// TIA Portal V17 export
// export: Created 2023-04-07T09:30:33.3999419Z, ExportSetting WithDefaults, DisplayName Totally Integrated Automation Portal, DisplayVersion V17 Update 4, DisplayName TIA Portal Openness, DisplayVersion V17 Update 4, DisplayName TIA Portal Version Control Interface, DisplayVersion V17, DisplayName STEP 7 Professional, DisplayVersion V17 Update 4, DisplayName STEP 7 Safety, DisplayVersion V17, DisplayName WinCC Professional, DisplayVersion V17 Update 4
FUNCTION "PCS Faults_1" : Void   // FC43, LAD
{ S7_Optimized_Access := 'TRUE' }
VERSION : 0.1
// stored: AutoNumber false, IsIECCheckEnabled false, SetENOAutomatically false, UDAEnableTagReadback false
   VAR_TEMP
      wMF1 : Word;
      wMF2 : Word;
      wMF3 : Word;
      wMF4 : Word;
      wMW1 : Word;
      wMW2 : Word;
      wMW3 : Word;
      wMW4 : Word;
   END_VAR
   VAR_TEMP   // added for the SCL form of the ladder/FBD networks
      _w1 : Bool;
      _w2 : Bool;
      _w3 : Bool;
      _w4 : Bool;
   END_VAR
BEGIN

REGION Network 1: Inverter Faults
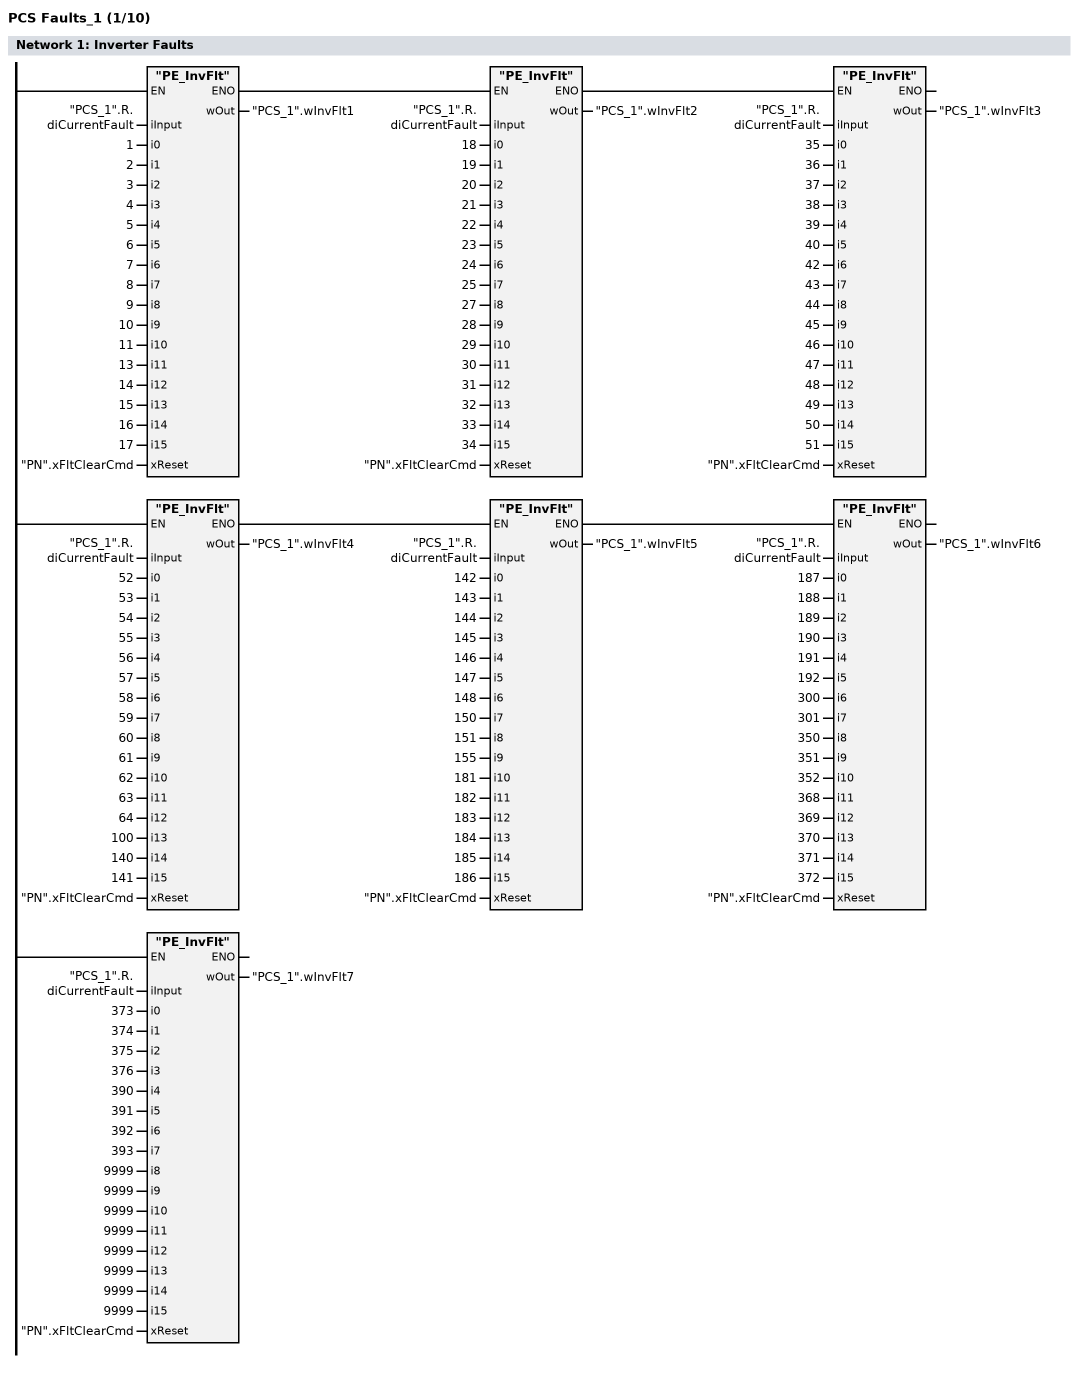
   RUNG wire#powerrail
      "PE_InvFlt"(iInput := "PCS_1".R.diCurrentFault, i0 := 1, i1 := 2, i2 := 3, i3 := 4, i4 := 5, i5 := 6, i6 := 7, i7 := 8, i8 := 9, i9 := 10, i10 := 11, i11 := 13, i12 := 14, i13 := 15, i14 := 16, i15 := 17, xReset := "PN".xFltClearCmd, wOut => "PCS_1".wInvFlt1)
      "PE_InvFlt"(iInput := "PCS_1".R.diCurrentFault, i0 := 18, i1 := 19, i2 := 20, i3 := 21, i4 := 22, i5 := 23, i6 := 24, i7 := 25, i8 := 27, i9 := 28, i10 := 29, i11 := 30, i12 := 31, i13 := 32, i14 := 33, i15 := 34, xReset := "PN".xFltClearCmd, wOut => "PCS_1".wInvFlt2)
      "PE_InvFlt"(iInput := "PCS_1".R.diCurrentFault, i0 := 35, i1 := 36, i2 := 37, i3 := 38, i4 := 39, i5 := 40, i6 := 42, i7 := 43, i8 := 44, i9 := 45, i10 := 46, i11 := 47, i12 := 48, i13 := 49, i14 := 50, i15 := 51, xReset := "PN".xFltClearCmd, wOut => "PCS_1".wInvFlt3)
   END_RUNG
   RUNG wire#powerrail
      "PE_InvFlt"(iInput := "PCS_1".R.diCurrentFault, i0 := 52, i1 := 53, i2 := 54, i3 := 55, i4 := 56, i5 := 57, i6 := 58, i7 := 59, i8 := 60, i9 := 61, i10 := 62, i11 := 63, i12 := 64, i13 := 100, i14 := 140, i15 := 141, xReset := "PN".xFltClearCmd, wOut => "PCS_1".wInvFlt4)
      "PE_InvFlt"(iInput := "PCS_1".R.diCurrentFault, i0 := 142, i1 := 143, i2 := 144, i3 := 145, i4 := 146, i5 := 147, i6 := 148, i7 := 150, i8 := 151, i9 := 155, i10 := 181, i11 := 182, i12 := 183, i13 := 184, i14 := 185, i15 := 186, xReset := "PN".xFltClearCmd, wOut => "PCS_1".wInvFlt5)
      "PE_InvFlt"(iInput := "PCS_1".R.diCurrentFault, i0 := 187, i1 := 188, i2 := 189, i3 := 190, i4 := 191, i5 := 192, i6 := 300, i7 := 301, i8 := 350, i9 := 351, i10 := 352, i11 := 368, i12 := 369, i13 := 370, i14 := 371, i15 := 372, xReset := "PN".xFltClearCmd, wOut => "PCS_1".wInvFlt6)
   END_RUNG
   RUNG wire#powerrail
      "PE_InvFlt"(iInput := "PCS_1".R.diCurrentFault, i0 := 373, i1 := 374, i2 := 375, i3 := 376, i4 := 390, i5 := 391, i6 := 392, i7 := 393, i8 := 9999, i9 := 9999, i10 := 9999, i11 := 9999, i12 := 9999, i13 := 9999, i14 := 9999, i15 := 9999, xReset := "PN".xFltClearCmd, wOut => "PCS_1".wInvFlt7)
   END_RUNG
   // the same network as SCL:
   "PE_InvFlt"(iInput := "PCS_1".R.diCurrentFault,
               i0 := 1,
               i1 := 2,
               i2 := 3,
               i3 := 4,
               i4 := 5,
               i5 := 6,
               i6 := 7,
               i7 := 8,
               i8 := 9,
               i9 := 10,
               i10 := 11,
               i11 := 13,
               i12 := 14,
               i13 := 15,
               i14 := 16,
               i15 := 17,
               xReset := "PN".xFltClearCmd,
               wOut => "PCS_1".wInvFlt1,
               ENO => #_w1);
   "PE_InvFlt"(EN := #_w1,
               iInput := "PCS_1".R.diCurrentFault,
               i0 := 18,
               i1 := 19,
               i2 := 20,
               i3 := 21,
               i4 := 22,
               i5 := 23,
               i6 := 24,
               i7 := 25,
               i8 := 27,
               i9 := 28,
               i10 := 29,
               i11 := 30,
               i12 := 31,
               i13 := 32,
               i14 := 33,
               i15 := 34,
               xReset := "PN".xFltClearCmd,
               wOut => "PCS_1".wInvFlt2,
               ENO => #_w2);
   IF #_w2 THEN
       "PE_InvFlt"(iInput := "PCS_1".R.diCurrentFault,
                   i0 := 35,
                   i1 := 36,
                   i2 := 37,
                   i3 := 38,
                   i4 := 39,
                   i5 := 40,
                   i6 := 42,
                   i7 := 43,
                   i8 := 44,
                   i9 := 45,
                   i10 := 46,
                   i11 := 47,
                   i12 := 48,
                   i13 := 49,
                   i14 := 50,
                   i15 := 51,
                   xReset := "PN".xFltClearCmd,
                   wOut => "PCS_1".wInvFlt3);
   END_IF;
   "PE_InvFlt"(iInput := "PCS_1".R.diCurrentFault,
               i0 := 52,
               i1 := 53,
               i2 := 54,
               i3 := 55,
               i4 := 56,
               i5 := 57,
               i6 := 58,
               i7 := 59,
               i8 := 60,
               i9 := 61,
               i10 := 62,
               i11 := 63,
               i12 := 64,
               i13 := 100,
               i14 := 140,
               i15 := 141,
               xReset := "PN".xFltClearCmd,
               wOut => "PCS_1".wInvFlt4,
               ENO => #_w3);
   "PE_InvFlt"(EN := #_w3,
               iInput := "PCS_1".R.diCurrentFault,
               i0 := 142,
               i1 := 143,
               i2 := 144,
               i3 := 145,
               i4 := 146,
               i5 := 147,
               i6 := 148,
               i7 := 150,
               i8 := 151,
               i9 := 155,
               i10 := 181,
               i11 := 182,
               i12 := 183,
               i13 := 184,
               i14 := 185,
               i15 := 186,
               xReset := "PN".xFltClearCmd,
               wOut => "PCS_1".wInvFlt5,
               ENO => #_w4);
   IF #_w4 THEN
       "PE_InvFlt"(iInput := "PCS_1".R.diCurrentFault,
                   i0 := 187,
                   i1 := 188,
                   i2 := 189,
                   i3 := 190,
                   i4 := 191,
                   i5 := 192,
                   i6 := 300,
                   i7 := 301,
                   i8 := 350,
                   i9 := 351,
                   i10 := 352,
                   i11 := 368,
                   i12 := 369,
                   i13 := 370,
                   i14 := 371,
                   i15 := 372,
                   xReset := "PN".xFltClearCmd,
                   wOut => "PCS_1".wInvFlt6);
   END_IF;
   "PE_InvFlt"(iInput := "PCS_1".R.diCurrentFault,
               i0 := 373,
               i1 := 374,
               i2 := 375,
               i3 := 376,
               i4 := 390,
               i5 := 391,
               i6 := 392,
               i7 := 393,
               i8 := 9999,
               i9 := 9999,
               i10 := 9999,
               i11 := 9999,
               i12 := 9999,
               i13 := 9999,
               i14 := 9999,
               i15 := 9999,
               xReset := "PN".xFltClearCmd,
               wOut => "PCS_1".wInvFlt7);
END_REGION

REGION Network 2: Inverter Warning
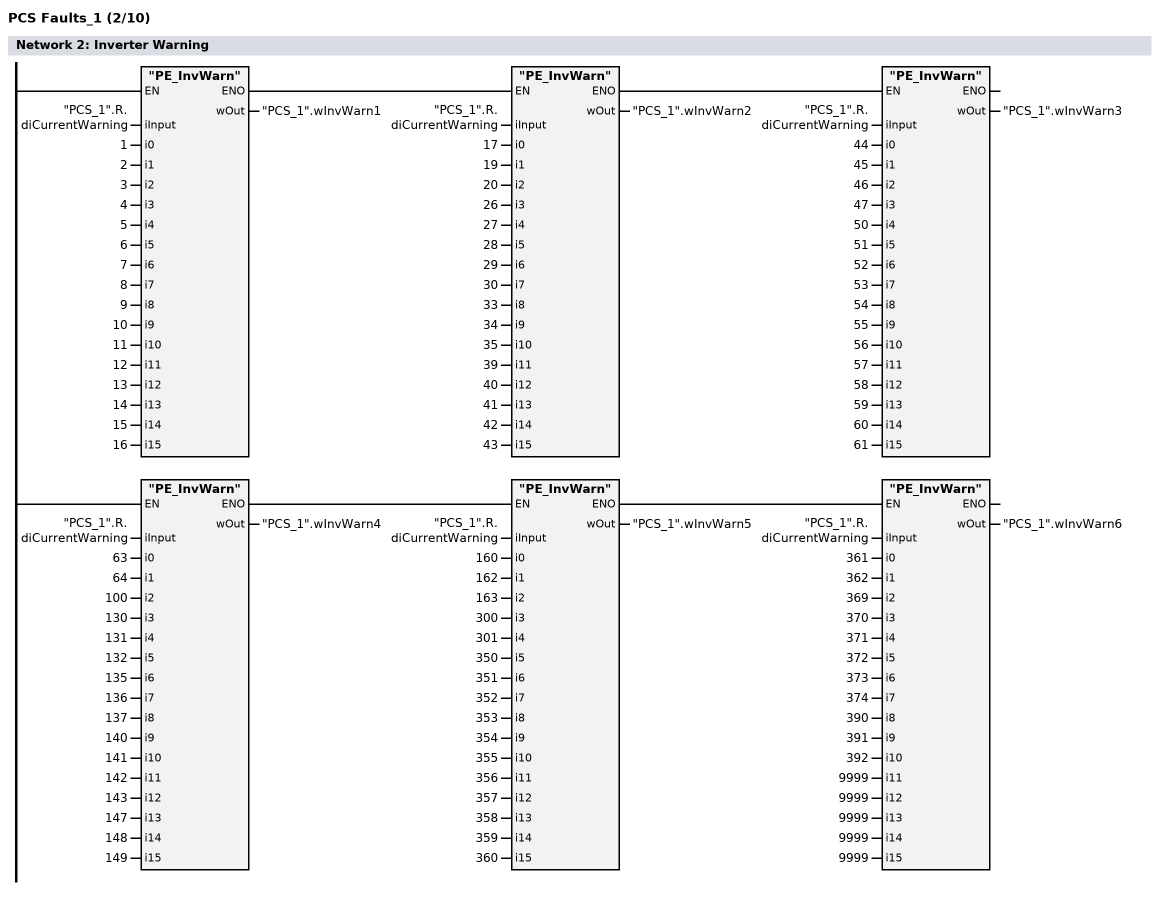
   RUNG wire#powerrail
      "PE_InvWarn"(iInput := "PCS_1".R.diCurrentWarning, i0 := 1, i1 := 2, i2 := 3, i3 := 4, i4 := 5, i5 := 6, i6 := 7, i7 := 8, i8 := 9, i9 := 10, i10 := 11, i11 := 12, i12 := 13, i13 := 14, i14 := 15, i15 := 16, wOut => "PCS_1".wInvWarn1)
      "PE_InvWarn"(iInput := "PCS_1".R.diCurrentWarning, i0 := 17, i1 := 19, i2 := 20, i3 := 26, i4 := 27, i5 := 28, i6 := 29, i7 := 30, i8 := 33, i9 := 34, i10 := 35, i11 := 39, i12 := 40, i13 := 41, i14 := 42, i15 := 43, wOut => "PCS_1".wInvWarn2)
      "PE_InvWarn"(iInput := "PCS_1".R.diCurrentWarning, i0 := 44, i1 := 45, i2 := 46, i3 := 47, i4 := 50, i5 := 51, i6 := 52, i7 := 53, i8 := 54, i9 := 55, i10 := 56, i11 := 57, i12 := 58, i13 := 59, i14 := 60, i15 := 61, wOut => "PCS_1".wInvWarn3)
   END_RUNG
   RUNG wire#powerrail
      "PE_InvWarn"(iInput := "PCS_1".R.diCurrentWarning, i0 := 63, i1 := 64, i2 := 100, i3 := 130, i4 := 131, i5 := 132, i6 := 135, i7 := 136, i8 := 137, i9 := 140, i10 := 141, i11 := 142, i12 := 143, i13 := 147, i14 := 148, i15 := 149, wOut => "PCS_1".wInvWarn4)
      "PE_InvWarn"(iInput := "PCS_1".R.diCurrentWarning, i0 := 160, i1 := 162, i2 := 163, i3 := 300, i4 := 301, i5 := 350, i6 := 351, i7 := 352, i8 := 353, i9 := 354, i10 := 355, i11 := 356, i12 := 357, i13 := 358, i14 := 359, i15 := 360, wOut => "PCS_1".wInvWarn5)
      "PE_InvWarn"(iInput := "PCS_1".R.diCurrentWarning, i0 := 361, i1 := 362, i2 := 369, i3 := 370, i4 := 371, i5 := 372, i6 := 373, i7 := 374, i8 := 390, i9 := 391, i10 := 392, i11 := 9999, i12 := 9999, i13 := 9999, i14 := 9999, i15 := 9999, wOut => "PCS_1".wInvWarn6)
   END_RUNG
   // the same network as SCL:
   "PE_InvWarn"(iInput := "PCS_1".R.diCurrentWarning,
                i0 := 1,
                i1 := 2,
                i2 := 3,
                i3 := 4,
                i4 := 5,
                i5 := 6,
                i6 := 7,
                i7 := 8,
                i8 := 9,
                i9 := 10,
                i10 := 11,
                i11 := 12,
                i12 := 13,
                i13 := 14,
                i14 := 15,
                i15 := 16,
                wOut => "PCS_1".wInvWarn1,
                ENO => #_w1);
   "PE_InvWarn"(EN := #_w1,
                iInput := "PCS_1".R.diCurrentWarning,
                i0 := 17,
                i1 := 19,
                i2 := 20,
                i3 := 26,
                i4 := 27,
                i5 := 28,
                i6 := 29,
                i7 := 30,
                i8 := 33,
                i9 := 34,
                i10 := 35,
                i11 := 39,
                i12 := 40,
                i13 := 41,
                i14 := 42,
                i15 := 43,
                wOut => "PCS_1".wInvWarn2,
                ENO => #_w2);
   IF #_w2 THEN
       "PE_InvWarn"(iInput := "PCS_1".R.diCurrentWarning,
                    i0 := 44,
                    i1 := 45,
                    i2 := 46,
                    i3 := 47,
                    i4 := 50,
                    i5 := 51,
                    i6 := 52,
                    i7 := 53,
                    i8 := 54,
                    i9 := 55,
                    i10 := 56,
                    i11 := 57,
                    i12 := 58,
                    i13 := 59,
                    i14 := 60,
                    i15 := 61,
                    wOut => "PCS_1".wInvWarn3);
   END_IF;
   "PE_InvWarn"(iInput := "PCS_1".R.diCurrentWarning,
                i0 := 63,
                i1 := 64,
                i2 := 100,
                i3 := 130,
                i4 := 131,
                i5 := 132,
                i6 := 135,
                i7 := 136,
                i8 := 137,
                i9 := 140,
                i10 := 141,
                i11 := 142,
                i12 := 143,
                i13 := 147,
                i14 := 148,
                i15 := 149,
                wOut => "PCS_1".wInvWarn4,
                ENO => #_w3);
   "PE_InvWarn"(EN := #_w3,
                iInput := "PCS_1".R.diCurrentWarning,
                i0 := 160,
                i1 := 162,
                i2 := 163,
                i3 := 300,
                i4 := 301,
                i5 := 350,
                i6 := 351,
                i7 := 352,
                i8 := 353,
                i9 := 354,
                i10 := 355,
                i11 := 356,
                i12 := 357,
                i13 := 358,
                i14 := 359,
                i15 := 360,
                wOut => "PCS_1".wInvWarn5,
                ENO => #_w4);
   IF #_w4 THEN
       "PE_InvWarn"(iInput := "PCS_1".R.diCurrentWarning,
                    i0 := 361,
                    i1 := 362,
                    i2 := 369,
                    i3 := 370,
                    i4 := 371,
                    i5 := 372,
                    i6 := 373,
                    i7 := 374,
                    i8 := 390,
                    i9 := 391,
                    i10 := 392,
                    i11 := 9999,
                    i12 := 9999,
                    i13 := 9999,
                    i14 := 9999,
                    i15 := 9999,
                    wOut => "PCS_1".wInvWarn6);
   END_IF;
END_REGION

REGION Network 3: Module Faults
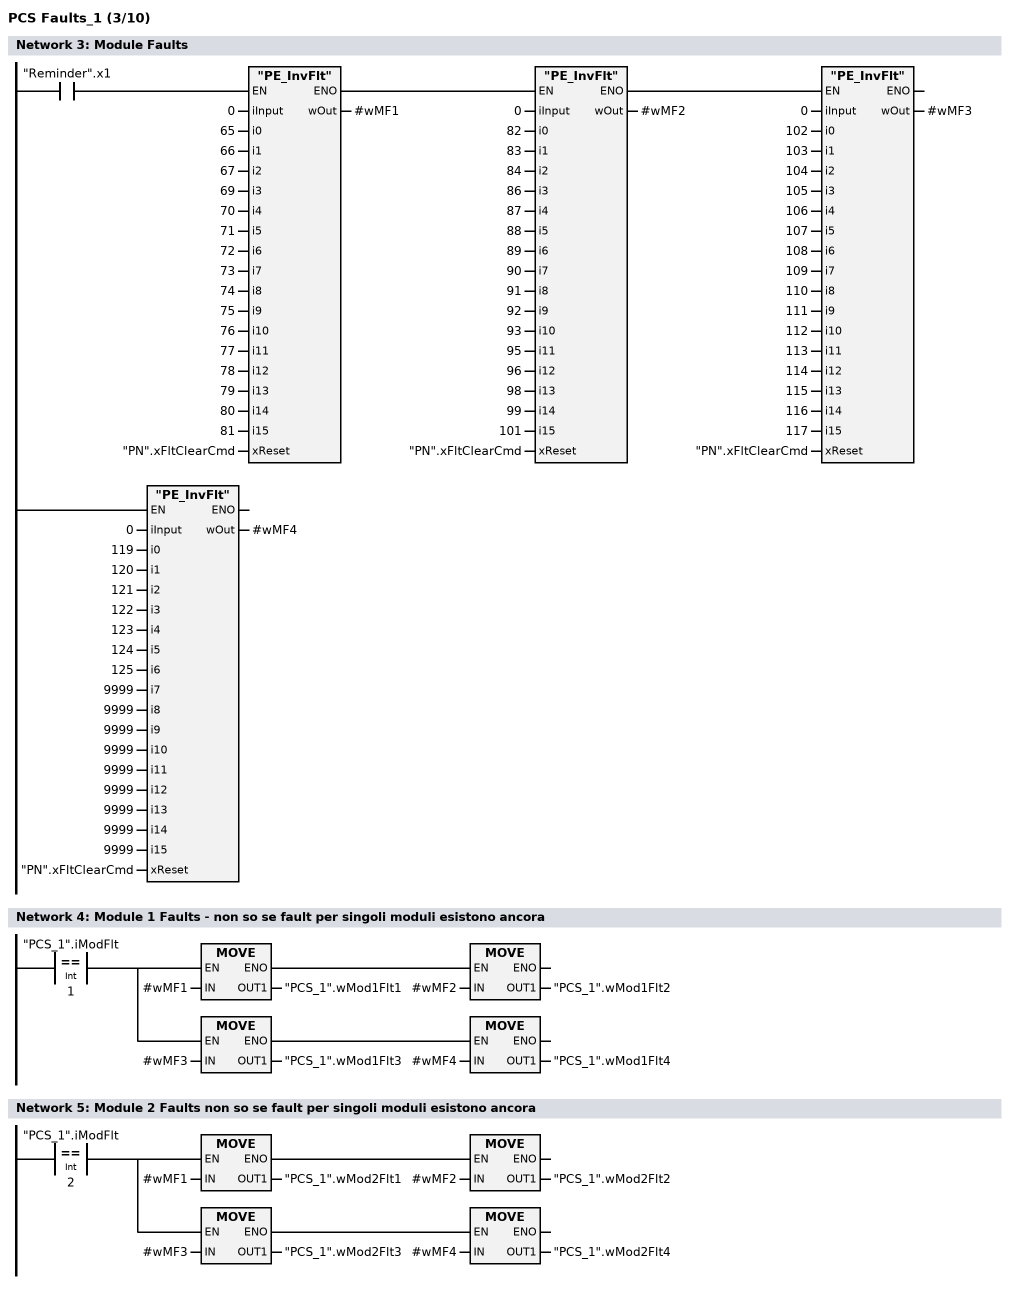
   RUNG wire#powerrail
      Contact( "Reminder".x1 )
      "PE_InvFlt"(iInput := 0, i0 := 65, i1 := 66, i2 := 67, i3 := 69, i4 := 70, i5 := 71, i6 := 72, i7 := 73, i8 := 74, i9 := 75, i10 := 76, i11 := 77, i12 := 78, i13 := 79, i14 := 80, i15 := 81, xReset := "PN".xFltClearCmd, wOut => #wMF1)
      "PE_InvFlt"(iInput := 0, i0 := 82, i1 := 83, i2 := 84, i3 := 86, i4 := 87, i5 := 88, i6 := 89, i7 := 90, i8 := 91, i9 := 92, i10 := 93, i11 := 95, i12 := 96, i13 := 98, i14 := 99, i15 := 101, xReset := "PN".xFltClearCmd, wOut => #wMF2)
      "PE_InvFlt"(iInput := 0, i0 := 102, i1 := 103, i2 := 104, i3 := 105, i4 := 106, i5 := 107, i6 := 108, i7 := 109, i8 := 110, i9 := 111, i10 := 112, i11 := 113, i12 := 114, i13 := 115, i14 := 116, i15 := 117, xReset := "PN".xFltClearCmd, wOut => #wMF3)
   END_RUNG
   RUNG wire#powerrail
      "PE_InvFlt"(iInput := 0, i0 := 119, i1 := 120, i2 := 121, i3 := 122, i4 := 123, i5 := 124, i6 := 125, i7 := 9999, i8 := 9999, i9 := 9999, i10 := 9999, i11 := 9999, i12 := 9999, i13 := 9999, i14 := 9999, i15 := 9999, xReset := "PN".xFltClearCmd, wOut => #wMF4)
   END_RUNG
   // the same network as SCL:
   "PE_InvFlt"(EN := "Reminder".x1,
               iInput := 0,
               i0 := 65,
               i1 := 66,
               i2 := 67,
               i3 := 69,
               i4 := 70,
               i5 := 71,
               i6 := 72,
               i7 := 73,
               i8 := 74,
               i9 := 75,
               i10 := 76,
               i11 := 77,
               i12 := 78,
               i13 := 79,
               i14 := 80,
               i15 := 81,
               xReset := "PN".xFltClearCmd,
               wOut => #wMF1,
               ENO => #_w1);
   "PE_InvFlt"(EN := #_w1,
               iInput := 0,
               i0 := 82,
               i1 := 83,
               i2 := 84,
               i3 := 86,
               i4 := 87,
               i5 := 88,
               i6 := 89,
               i7 := 90,
               i8 := 91,
               i9 := 92,
               i10 := 93,
               i11 := 95,
               i12 := 96,
               i13 := 98,
               i14 := 99,
               i15 := 101,
               xReset := "PN".xFltClearCmd,
               wOut => #wMF2,
               ENO => #_w2);
   IF #_w2 THEN
       "PE_InvFlt"(iInput := 0,
                   i0 := 102,
                   i1 := 103,
                   i2 := 104,
                   i3 := 105,
                   i4 := 106,
                   i5 := 107,
                   i6 := 108,
                   i7 := 109,
                   i8 := 110,
                   i9 := 111,
                   i10 := 112,
                   i11 := 113,
                   i12 := 114,
                   i13 := 115,
                   i14 := 116,
                   i15 := 117,
                   xReset := "PN".xFltClearCmd,
                   wOut => #wMF3);
   END_IF;
   "PE_InvFlt"(iInput := 0,
               i0 := 119,
               i1 := 120,
               i2 := 121,
               i3 := 122,
               i4 := 123,
               i5 := 124,
               i6 := 125,
               i7 := 9999,
               i8 := 9999,
               i9 := 9999,
               i10 := 9999,
               i11 := 9999,
               i12 := 9999,
               i13 := 9999,
               i14 := 9999,
               i15 := 9999,
               xReset := "PN".xFltClearCmd,
               wOut => #wMF4);
END_REGION

REGION Network 4: Module 1 Faults - non so se fault per singoli moduli esistono ancora
   RUNG wire#powerrail
      { S7_Templates := "SrcType := Int" } EQ_Contact(in1 := "PCS_1".iModFlt, in2 := 1)
      wire#w1
      Move(in := #wMF1, out1 => "PCS_1".wMod1Flt1)
      Move(in := #wMF2, out1 => "PCS_1".wMod1Flt2)
   END_RUNG
   RUNG wire#w1
      Move(in := #wMF3, out1 => "PCS_1".wMod1Flt3)
      Move(in := #wMF4, out1 => "PCS_1".wMod1Flt4)
   END_RUNG
   // the same network as SCL:
   IF "PCS_1".iModFlt = 1 THEN
       "PCS_1".wMod1Flt1 := #wMF1;
       "PCS_1".wMod1Flt2 := #wMF2;
       "PCS_1".wMod1Flt3 := #wMF3;
       "PCS_1".wMod1Flt4 := #wMF4;
   END_IF;
END_REGION

REGION Network 5: Module 2 Faults non so se fault per singoli moduli esistono ancora
   RUNG wire#powerrail
      { S7_Templates := "SrcType := Int" } EQ_Contact(in1 := "PCS_1".iModFlt, in2 := 2)
      wire#w1
      Move(in := #wMF1, out1 => "PCS_1".wMod2Flt1)
      Move(in := #wMF2, out1 => "PCS_1".wMod2Flt2)
   END_RUNG
   RUNG wire#w1
      Move(in := #wMF3, out1 => "PCS_1".wMod2Flt3)
      Move(in := #wMF4, out1 => "PCS_1".wMod2Flt4)
   END_RUNG
   // the same network as SCL:
   IF "PCS_1".iModFlt = 2 THEN
       "PCS_1".wMod2Flt1 := #wMF1;
       "PCS_1".wMod2Flt2 := #wMF2;
       "PCS_1".wMod2Flt3 := #wMF3;
       "PCS_1".wMod2Flt4 := #wMF4;
   END_IF;
END_REGION

REGION Network 6: Module 3 Faults
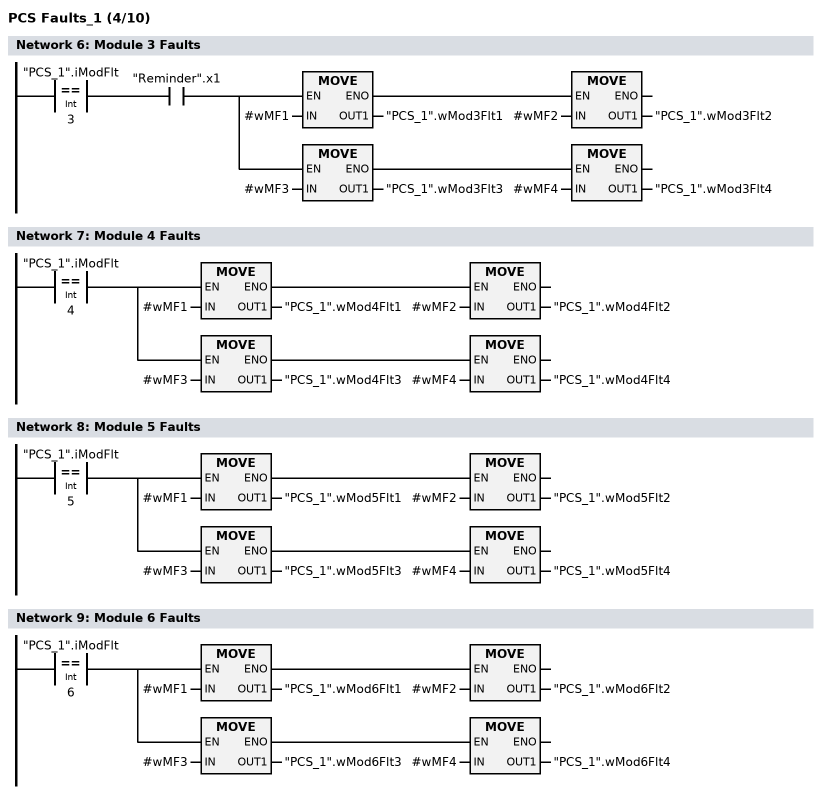
   RUNG wire#powerrail
      { S7_Templates := "SrcType := Int" } EQ_Contact(in1 := "PCS_1".iModFlt, in2 := 3)
      Contact( "Reminder".x1 )
      wire#w1
      Move(in := #wMF1, out1 => "PCS_1".wMod3Flt1)
      Move(in := #wMF2, out1 => "PCS_1".wMod3Flt2)
   END_RUNG
   RUNG wire#w1
      Move(in := #wMF3, out1 => "PCS_1".wMod3Flt3)
      Move(in := #wMF4, out1 => "PCS_1".wMod3Flt4)
   END_RUNG
   // the same network as SCL:
   IF ("PCS_1".iModFlt = 3) AND "Reminder".x1 THEN
       "PCS_1".wMod3Flt1 := #wMF1;
       "PCS_1".wMod3Flt2 := #wMF2;
       "PCS_1".wMod3Flt3 := #wMF3;
       "PCS_1".wMod3Flt4 := #wMF4;
   END_IF;
END_REGION

REGION Network 7: Module 4 Faults
   RUNG wire#powerrail
      { S7_Templates := "SrcType := Int" } EQ_Contact(in1 := "PCS_1".iModFlt, in2 := 4)
      wire#w1
      Move(in := #wMF1, out1 => "PCS_1".wMod4Flt1)
      Move(in := #wMF2, out1 => "PCS_1".wMod4Flt2)
   END_RUNG
   RUNG wire#w1
      Move(in := #wMF3, out1 => "PCS_1".wMod4Flt3)
      Move(in := #wMF4, out1 => "PCS_1".wMod4Flt4)
   END_RUNG
   // the same network as SCL:
   IF "PCS_1".iModFlt = 4 THEN
       "PCS_1".wMod4Flt1 := #wMF1;
       "PCS_1".wMod4Flt2 := #wMF2;
       "PCS_1".wMod4Flt3 := #wMF3;
       "PCS_1".wMod4Flt4 := #wMF4;
   END_IF;
END_REGION

REGION Network 8: Module 5 Faults
   RUNG wire#powerrail
      { S7_Templates := "SrcType := Int" } EQ_Contact(in1 := "PCS_1".iModFlt, in2 := 5)
      wire#w1
      Move(in := #wMF1, out1 => "PCS_1".wMod5Flt1)
      Move(in := #wMF2, out1 => "PCS_1".wMod5Flt2)
   END_RUNG
   RUNG wire#w1
      Move(in := #wMF3, out1 => "PCS_1".wMod5Flt3)
      Move(in := #wMF4, out1 => "PCS_1".wMod5Flt4)
   END_RUNG
   // the same network as SCL:
   IF "PCS_1".iModFlt = 5 THEN
       "PCS_1".wMod5Flt1 := #wMF1;
       "PCS_1".wMod5Flt2 := #wMF2;
       "PCS_1".wMod5Flt3 := #wMF3;
       "PCS_1".wMod5Flt4 := #wMF4;
   END_IF;
END_REGION

REGION Network 9: Module 6 Faults
   RUNG wire#powerrail
      { S7_Templates := "SrcType := Int" } EQ_Contact(in1 := "PCS_1".iModFlt, in2 := 6)
      wire#w1
      Move(in := #wMF1, out1 => "PCS_1".wMod6Flt1)
      Move(in := #wMF2, out1 => "PCS_1".wMod6Flt2)
   END_RUNG
   RUNG wire#w1
      Move(in := #wMF3, out1 => "PCS_1".wMod6Flt3)
      Move(in := #wMF4, out1 => "PCS_1".wMod6Flt4)
   END_RUNG
   // the same network as SCL:
   IF "PCS_1".iModFlt = 6 THEN
       "PCS_1".wMod6Flt1 := #wMF1;
       "PCS_1".wMod6Flt2 := #wMF2;
       "PCS_1".wMod6Flt3 := #wMF3;
       "PCS_1".wMod6Flt4 := #wMF4;
   END_IF;
END_REGION

REGION Network 10: Module Warnings
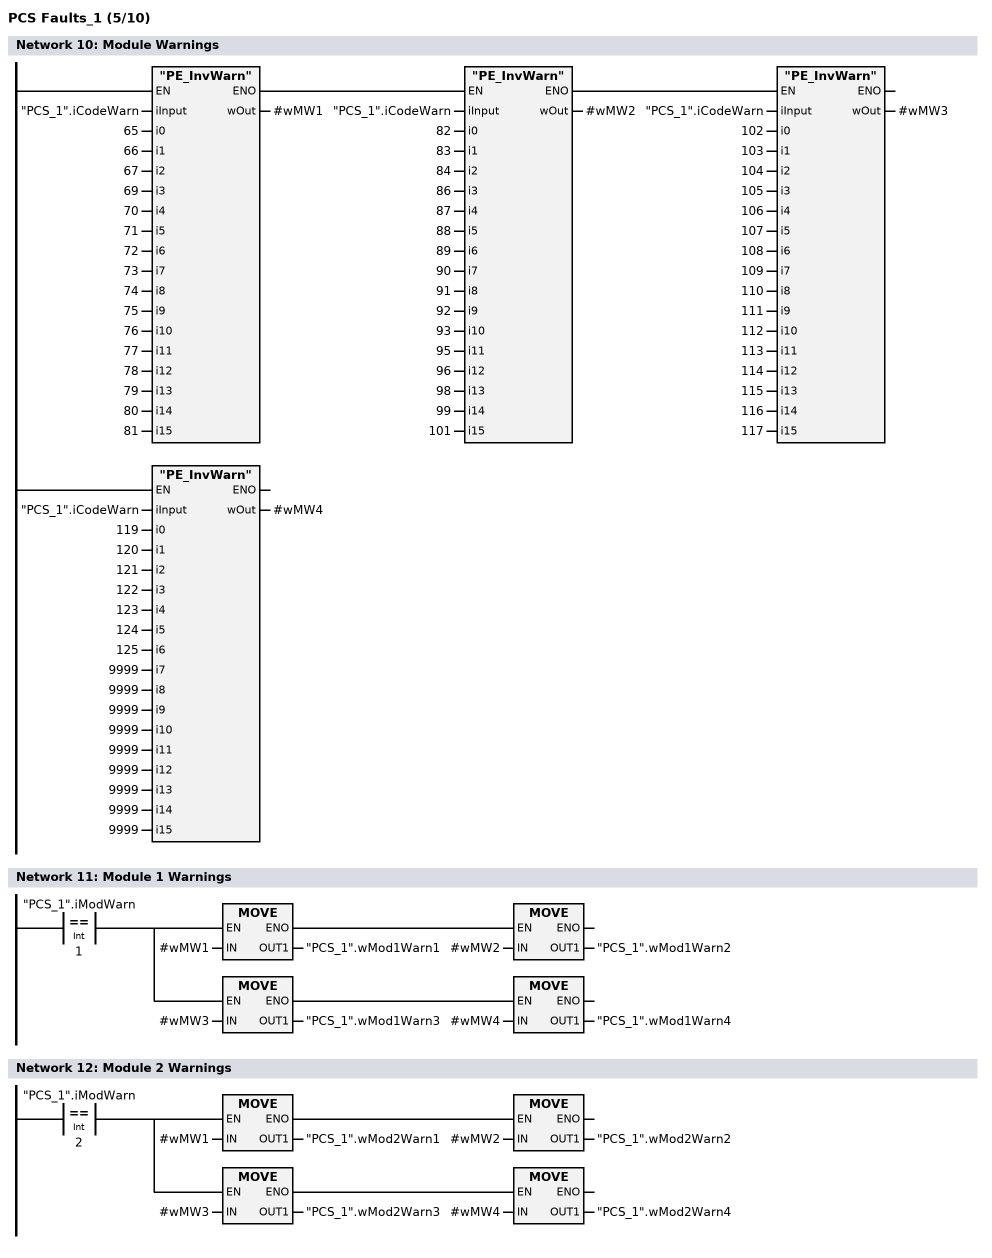
   RUNG wire#powerrail
      "PE_InvWarn"(iInput := "PCS_1".iCodeWarn, i0 := 65, i1 := 66, i2 := 67, i3 := 69, i4 := 70, i5 := 71, i6 := 72, i7 := 73, i8 := 74, i9 := 75, i10 := 76, i11 := 77, i12 := 78, i13 := 79, i14 := 80, i15 := 81, wOut => #wMW1)
      "PE_InvWarn"(iInput := "PCS_1".iCodeWarn, i0 := 82, i1 := 83, i2 := 84, i3 := 86, i4 := 87, i5 := 88, i6 := 89, i7 := 90, i8 := 91, i9 := 92, i10 := 93, i11 := 95, i12 := 96, i13 := 98, i14 := 99, i15 := 101, wOut => #wMW2)
      "PE_InvWarn"(iInput := "PCS_1".iCodeWarn, i0 := 102, i1 := 103, i2 := 104, i3 := 105, i4 := 106, i5 := 107, i6 := 108, i7 := 109, i8 := 110, i9 := 111, i10 := 112, i11 := 113, i12 := 114, i13 := 115, i14 := 116, i15 := 117, wOut => #wMW3)
   END_RUNG
   RUNG wire#powerrail
      "PE_InvWarn"(iInput := "PCS_1".iCodeWarn, i0 := 119, i1 := 120, i2 := 121, i3 := 122, i4 := 123, i5 := 124, i6 := 125, i7 := 9999, i8 := 9999, i9 := 9999, i10 := 9999, i11 := 9999, i12 := 9999, i13 := 9999, i14 := 9999, i15 := 9999, wOut => #wMW4)
   END_RUNG
   // the same network as SCL:
   "PE_InvWarn"(iInput := "PCS_1".iCodeWarn,
                i0 := 65,
                i1 := 66,
                i2 := 67,
                i3 := 69,
                i4 := 70,
                i5 := 71,
                i6 := 72,
                i7 := 73,
                i8 := 74,
                i9 := 75,
                i10 := 76,
                i11 := 77,
                i12 := 78,
                i13 := 79,
                i14 := 80,
                i15 := 81,
                wOut => #wMW1,
                ENO => #_w1);
   "PE_InvWarn"(EN := #_w1,
                iInput := "PCS_1".iCodeWarn,
                i0 := 82,
                i1 := 83,
                i2 := 84,
                i3 := 86,
                i4 := 87,
                i5 := 88,
                i6 := 89,
                i7 := 90,
                i8 := 91,
                i9 := 92,
                i10 := 93,
                i11 := 95,
                i12 := 96,
                i13 := 98,
                i14 := 99,
                i15 := 101,
                wOut => #wMW2,
                ENO => #_w2);
   IF #_w2 THEN
       "PE_InvWarn"(iInput := "PCS_1".iCodeWarn,
                    i0 := 102,
                    i1 := 103,
                    i2 := 104,
                    i3 := 105,
                    i4 := 106,
                    i5 := 107,
                    i6 := 108,
                    i7 := 109,
                    i8 := 110,
                    i9 := 111,
                    i10 := 112,
                    i11 := 113,
                    i12 := 114,
                    i13 := 115,
                    i14 := 116,
                    i15 := 117,
                    wOut => #wMW3);
   END_IF;
   "PE_InvWarn"(iInput := "PCS_1".iCodeWarn,
                i0 := 119,
                i1 := 120,
                i2 := 121,
                i3 := 122,
                i4 := 123,
                i5 := 124,
                i6 := 125,
                i7 := 9999,
                i8 := 9999,
                i9 := 9999,
                i10 := 9999,
                i11 := 9999,
                i12 := 9999,
                i13 := 9999,
                i14 := 9999,
                i15 := 9999,
                wOut => #wMW4);
END_REGION

REGION Network 11: Module 1 Warnings
   RUNG wire#powerrail
      { S7_Templates := "SrcType := Int" } EQ_Contact(in1 := "PCS_1".iModWarn, in2 := 1)
      wire#w1
      Move(in := #wMW1, out1 => "PCS_1".wMod1Warn1)
      Move(in := #wMW2, out1 => "PCS_1".wMod1Warn2)
   END_RUNG
   RUNG wire#w1
      Move(in := #wMW3, out1 => "PCS_1".wMod1Warn3)
      Move(in := #wMW4, out1 => "PCS_1".wMod1Warn4)
   END_RUNG
   // the same network as SCL:
   IF "PCS_1".iModWarn = 1 THEN
       "PCS_1".wMod1Warn1 := #wMW1;
       "PCS_1".wMod1Warn2 := #wMW2;
       "PCS_1".wMod1Warn3 := #wMW3;
       "PCS_1".wMod1Warn4 := #wMW4;
   END_IF;
END_REGION

REGION Network 12: Module 2 Warnings
   RUNG wire#powerrail
      { S7_Templates := "SrcType := Int" } EQ_Contact(in1 := "PCS_1".iModWarn, in2 := 2)
      wire#w1
      Move(in := #wMW1, out1 => "PCS_1".wMod2Warn1)
      Move(in := #wMW2, out1 => "PCS_1".wMod2Warn2)
   END_RUNG
   RUNG wire#w1
      Move(in := #wMW3, out1 => "PCS_1".wMod2Warn3)
      Move(in := #wMW4, out1 => "PCS_1".wMod2Warn4)
   END_RUNG
   // the same network as SCL:
   IF "PCS_1".iModWarn = 2 THEN
       "PCS_1".wMod2Warn1 := #wMW1;
       "PCS_1".wMod2Warn2 := #wMW2;
       "PCS_1".wMod2Warn3 := #wMW3;
       "PCS_1".wMod2Warn4 := #wMW4;
   END_IF;
END_REGION

REGION Network 13: Module 3 Warnings
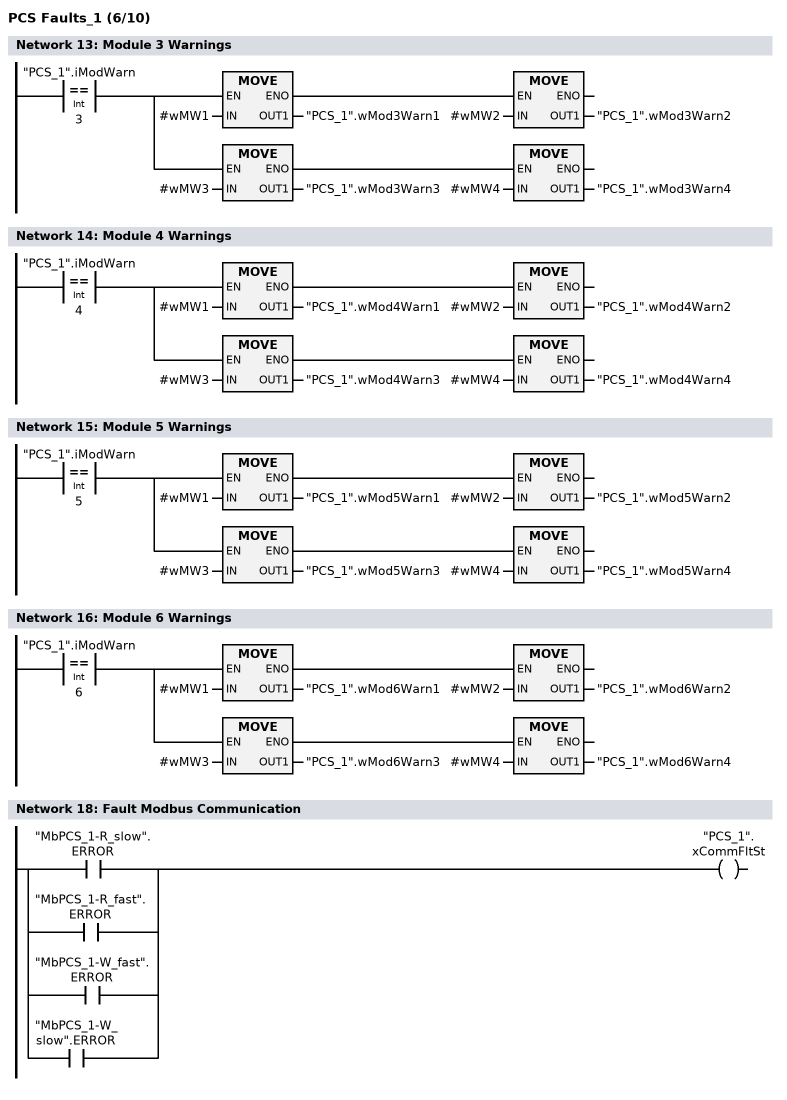
   RUNG wire#powerrail
      { S7_Templates := "SrcType := Int" } EQ_Contact(in1 := "PCS_1".iModWarn, in2 := 3)
      wire#w1
      Move(in := #wMW1, out1 => "PCS_1".wMod3Warn1)
      Move(in := #wMW2, out1 => "PCS_1".wMod3Warn2)
   END_RUNG
   RUNG wire#w1
      Move(in := #wMW3, out1 => "PCS_1".wMod3Warn3)
      Move(in := #wMW4, out1 => "PCS_1".wMod3Warn4)
   END_RUNG
   // the same network as SCL:
   IF "PCS_1".iModWarn = 3 THEN
       "PCS_1".wMod3Warn1 := #wMW1;
       "PCS_1".wMod3Warn2 := #wMW2;
       "PCS_1".wMod3Warn3 := #wMW3;
       "PCS_1".wMod3Warn4 := #wMW4;
   END_IF;
END_REGION

REGION Network 14: Module 4 Warnings
   RUNG wire#powerrail
      { S7_Templates := "SrcType := Int" } EQ_Contact(in1 := "PCS_1".iModWarn, in2 := 4)
      wire#w1
      Move(in := #wMW1, out1 => "PCS_1".wMod4Warn1)
      Move(in := #wMW2, out1 => "PCS_1".wMod4Warn2)
   END_RUNG
   RUNG wire#w1
      Move(in := #wMW3, out1 => "PCS_1".wMod4Warn3)
      Move(in := #wMW4, out1 => "PCS_1".wMod4Warn4)
   END_RUNG
   // the same network as SCL:
   IF "PCS_1".iModWarn = 4 THEN
       "PCS_1".wMod4Warn1 := #wMW1;
       "PCS_1".wMod4Warn2 := #wMW2;
       "PCS_1".wMod4Warn3 := #wMW3;
       "PCS_1".wMod4Warn4 := #wMW4;
   END_IF;
END_REGION

REGION Network 15: Module 5 Warnings
   RUNG wire#powerrail
      { S7_Templates := "SrcType := Int" } EQ_Contact(in1 := "PCS_1".iModWarn, in2 := 5)
      wire#w1
      Move(in := #wMW1, out1 => "PCS_1".wMod5Warn1)
      Move(in := #wMW2, out1 => "PCS_1".wMod5Warn2)
   END_RUNG
   RUNG wire#w1
      Move(in := #wMW3, out1 => "PCS_1".wMod5Warn3)
      Move(in := #wMW4, out1 => "PCS_1".wMod5Warn4)
   END_RUNG
   // the same network as SCL:
   IF "PCS_1".iModWarn = 5 THEN
       "PCS_1".wMod5Warn1 := #wMW1;
       "PCS_1".wMod5Warn2 := #wMW2;
       "PCS_1".wMod5Warn3 := #wMW3;
       "PCS_1".wMod5Warn4 := #wMW4;
   END_IF;
END_REGION

REGION Network 16: Module 6 Warnings
   RUNG wire#powerrail
      { S7_Templates := "SrcType := Int" } EQ_Contact(in1 := "PCS_1".iModWarn, in2 := 6)
      wire#w1
      Move(in := #wMW1, out1 => "PCS_1".wMod6Warn1)
      Move(in := #wMW2, out1 => "PCS_1".wMod6Warn2)
   END_RUNG
   RUNG wire#w1
      Move(in := #wMW3, out1 => "PCS_1".wMod6Warn3)
      Move(in := #wMW4, out1 => "PCS_1".wMod6Warn4)
   END_RUNG
   // the same network as SCL:
   IF "PCS_1".iModWarn = 6 THEN
       "PCS_1".wMod6Warn1 := #wMW1;
       "PCS_1".wMod6Warn2 := #wMW2;
       "PCS_1".wMod6Warn3 := #wMW3;
       "PCS_1".wMod6Warn4 := #wMW4;
   END_IF;
END_REGION

REGION Network 18: Fault Modbus Communication
   RUNG wire#powerrail
      Contact( "MbPCS_1-R_slow".ERROR )
      wire#w1
      Coil( "PCS_1".xCommFltSt )
   END_RUNG
   RUNG wire#powerrail
      Contact( "MbPCS_1-R_fast".ERROR )
   END_RUNG wire#w1
   RUNG wire#powerrail
      Contact( "MbPCS_1-W_fast".ERROR )
   END_RUNG wire#w1
   RUNG wire#powerrail
      Contact( "MbPCS_1-W_slow".ERROR )
   END_RUNG wire#w1
   // the same network as SCL:
   "PCS_1".xCommFltSt := "MbPCS_1-R_slow".ERROR OR "MbPCS_1-R_fast".ERROR OR "MbPCS_1-W_fast".ERROR OR "MbPCS_1-W_slow".ERROR;
END_REGION

REGION Network 19: Inverter Fault
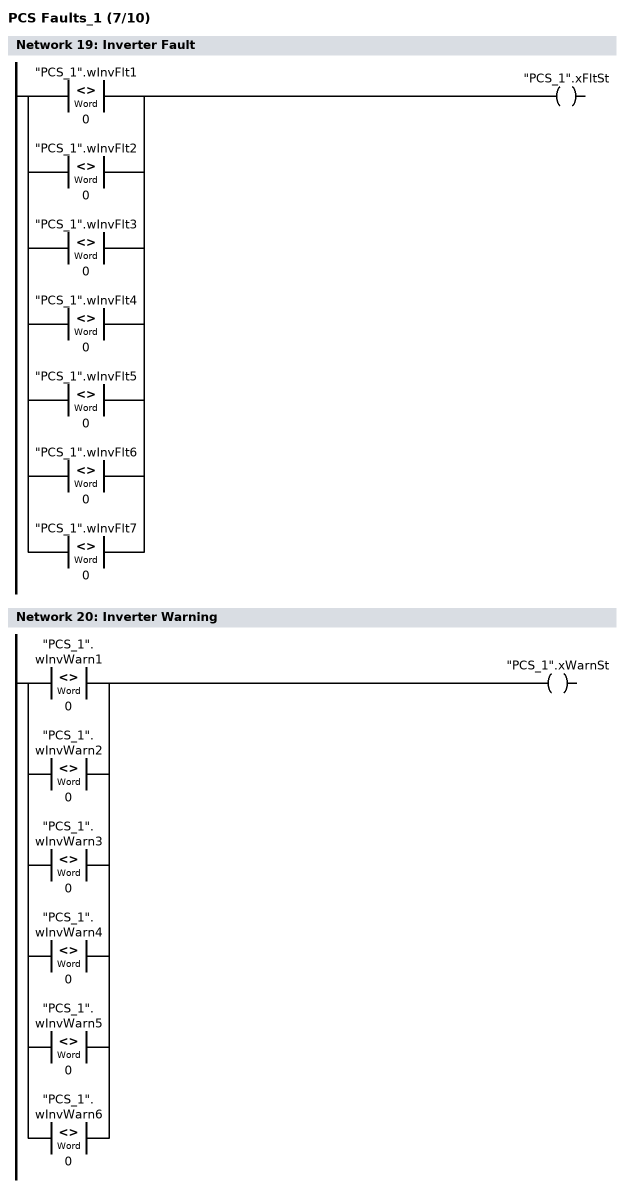
   RUNG wire#powerrail
      { S7_Templates := "SrcType := Word" } NE_Contact(in1 := "PCS_1".wInvFlt1, in2 := 0)
      wire#w1
      Coil( "PCS_1".xFltSt )
   END_RUNG
   RUNG wire#powerrail
      { S7_Templates := "SrcType := Word" } NE_Contact(in1 := "PCS_1".wInvFlt2, in2 := 0)
   END_RUNG wire#w1
   RUNG wire#powerrail
      { S7_Templates := "SrcType := Word" } NE_Contact(in1 := "PCS_1".wInvFlt3, in2 := 0)
   END_RUNG wire#w1
   RUNG wire#powerrail
      { S7_Templates := "SrcType := Word" } NE_Contact(in1 := "PCS_1".wInvFlt4, in2 := 0)
   END_RUNG wire#w1
   RUNG wire#powerrail
      { S7_Templates := "SrcType := Word" } NE_Contact(in1 := "PCS_1".wInvFlt5, in2 := 0)
   END_RUNG wire#w1
   RUNG wire#powerrail
      { S7_Templates := "SrcType := Word" } NE_Contact(in1 := "PCS_1".wInvFlt6, in2 := 0)
   END_RUNG wire#w1
   RUNG wire#powerrail
      { S7_Templates := "SrcType := Word" } NE_Contact(in1 := "PCS_1".wInvFlt7, in2 := 0)
   END_RUNG wire#w1
   // the same network as SCL:
   "PCS_1".xFltSt := ("PCS_1".wInvFlt1 <> 0) OR ("PCS_1".wInvFlt2 <> 0) OR ("PCS_1".wInvFlt3 <> 0) OR ("PCS_1".wInvFlt4 <> 0) OR ("PCS_1".wInvFlt5 <> 0) OR ("PCS_1".wInvFlt6 <> 0) OR ("PCS_1".wInvFlt7 <> 0);
END_REGION

REGION Network 20: Inverter Warning
   RUNG wire#powerrail
      { S7_Templates := "SrcType := Word" } NE_Contact(in1 := "PCS_1".wInvWarn1, in2 := 0)
      wire#w1
      Coil( "PCS_1".xWarnSt )
   END_RUNG
   RUNG wire#powerrail
      { S7_Templates := "SrcType := Word" } NE_Contact(in1 := "PCS_1".wInvWarn2, in2 := 0)
   END_RUNG wire#w1
   RUNG wire#powerrail
      { S7_Templates := "SrcType := Word" } NE_Contact(in1 := "PCS_1".wInvWarn3, in2 := 0)
   END_RUNG wire#w1
   RUNG wire#powerrail
      { S7_Templates := "SrcType := Word" } NE_Contact(in1 := "PCS_1".wInvWarn4, in2 := 0)
   END_RUNG wire#w1
   RUNG wire#powerrail
      { S7_Templates := "SrcType := Word" } NE_Contact(in1 := "PCS_1".wInvWarn5, in2 := 0)
   END_RUNG wire#w1
   RUNG wire#powerrail
      { S7_Templates := "SrcType := Word" } NE_Contact(in1 := "PCS_1".wInvWarn6, in2 := 0)
   END_RUNG wire#w1
   // the same network as SCL:
   "PCS_1".xWarnSt := ("PCS_1".wInvWarn1 <> 0) OR ("PCS_1".wInvWarn2 <> 0) OR ("PCS_1".wInvWarn3 <> 0) OR ("PCS_1".wInvWarn4 <> 0) OR ("PCS_1".wInvWarn5 <> 0) OR ("PCS_1".wInvWarn6 <> 0);
END_REGION

REGION Network 21: Da qua in poi è da chiarire se ci sono warninig e fault relativi ai moduli
END_REGION

REGION Network 22: Bus 1 Mod Fault -> Inizio OLD
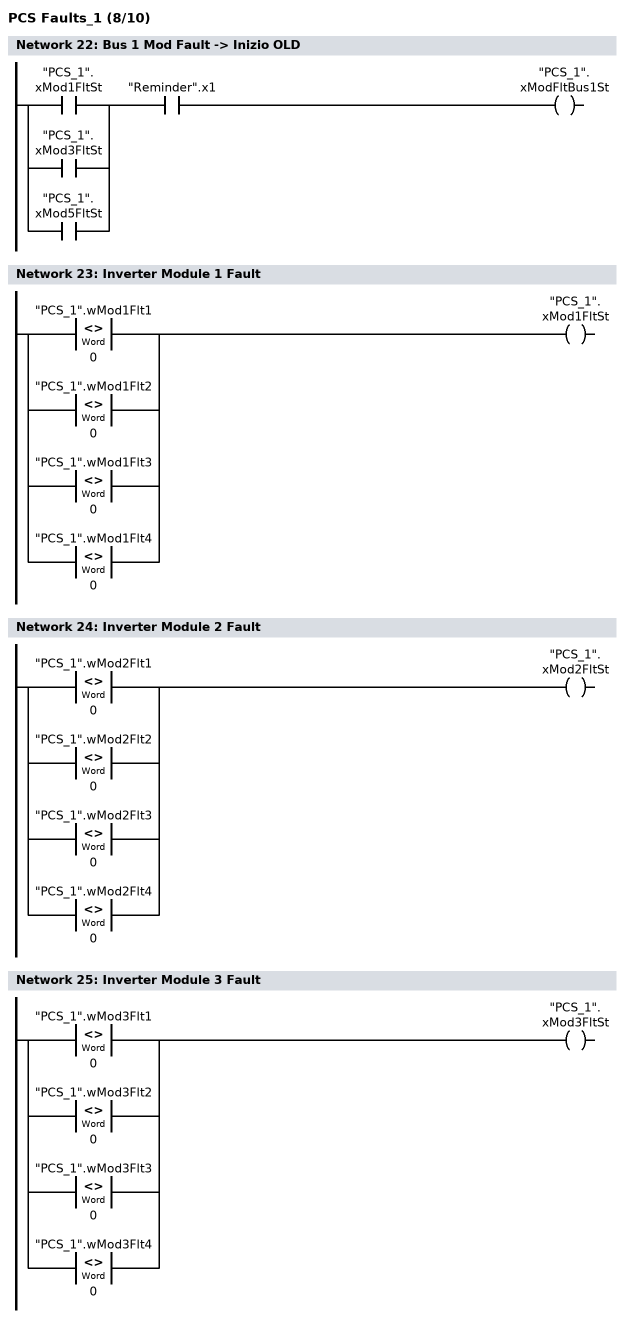
   RUNG wire#powerrail
      Contact( "PCS_1".xMod1FltSt )
      wire#w1
      Contact( "Reminder".x1 )
      Coil( "PCS_1".xModFltBus1St )
   END_RUNG
   RUNG wire#powerrail
      Contact( "PCS_1".xMod3FltSt )
   END_RUNG wire#w1
   RUNG wire#powerrail
      Contact( "PCS_1".xMod5FltSt )
   END_RUNG wire#w1
   // the same network as SCL:
   "PCS_1".xModFltBus1St := ("PCS_1".xMod1FltSt OR "PCS_1".xMod3FltSt OR "PCS_1".xMod5FltSt) AND "Reminder".x1;
END_REGION

REGION Network 23: Inverter Module 1 Fault
   RUNG wire#powerrail
      { S7_Templates := "SrcType := Word" } NE_Contact(in1 := "PCS_1".wMod1Flt1, in2 := 0)
      wire#w1
      Coil( "PCS_1".xMod1FltSt )
   END_RUNG
   RUNG wire#powerrail
      { S7_Templates := "SrcType := Word" } NE_Contact(in1 := "PCS_1".wMod1Flt2, in2 := 0)
   END_RUNG wire#w1
   RUNG wire#powerrail
      { S7_Templates := "SrcType := Word" } NE_Contact(in1 := "PCS_1".wMod1Flt3, in2 := 0)
   END_RUNG wire#w1
   RUNG wire#powerrail
      { S7_Templates := "SrcType := Word" } NE_Contact(in1 := "PCS_1".wMod1Flt4, in2 := 0)
   END_RUNG wire#w1
   // the same network as SCL:
   "PCS_1".xMod1FltSt := ("PCS_1".wMod1Flt1 <> 0) OR ("PCS_1".wMod1Flt2 <> 0) OR ("PCS_1".wMod1Flt3 <> 0) OR ("PCS_1".wMod1Flt4 <> 0);
END_REGION

REGION Network 24: Inverter Module 2 Fault
   RUNG wire#powerrail
      { S7_Templates := "SrcType := Word" } NE_Contact(in1 := "PCS_1".wMod2Flt1, in2 := 0)
      wire#w1
      Coil( "PCS_1".xMod2FltSt )
   END_RUNG
   RUNG wire#powerrail
      { S7_Templates := "SrcType := Word" } NE_Contact(in1 := "PCS_1".wMod2Flt2, in2 := 0)
   END_RUNG wire#w1
   RUNG wire#powerrail
      { S7_Templates := "SrcType := Word" } NE_Contact(in1 := "PCS_1".wMod2Flt3, in2 := 0)
   END_RUNG wire#w1
   RUNG wire#powerrail
      { S7_Templates := "SrcType := Word" } NE_Contact(in1 := "PCS_1".wMod2Flt4, in2 := 0)
   END_RUNG wire#w1
   // the same network as SCL:
   "PCS_1".xMod2FltSt := ("PCS_1".wMod2Flt1 <> 0) OR ("PCS_1".wMod2Flt2 <> 0) OR ("PCS_1".wMod2Flt3 <> 0) OR ("PCS_1".wMod2Flt4 <> 0);
END_REGION

REGION Network 25: Inverter Module 3 Fault
   RUNG wire#powerrail
      { S7_Templates := "SrcType := Word" } NE_Contact(in1 := "PCS_1".wMod3Flt1, in2 := 0)
      wire#w1
      Coil( "PCS_1".xMod3FltSt )
   END_RUNG
   RUNG wire#powerrail
      { S7_Templates := "SrcType := Word" } NE_Contact(in1 := "PCS_1".wMod3Flt2, in2 := 0)
   END_RUNG wire#w1
   RUNG wire#powerrail
      { S7_Templates := "SrcType := Word" } NE_Contact(in1 := "PCS_1".wMod3Flt3, in2 := 0)
   END_RUNG wire#w1
   RUNG wire#powerrail
      { S7_Templates := "SrcType := Word" } NE_Contact(in1 := "PCS_1".wMod3Flt4, in2 := 0)
   END_RUNG wire#w1
   // the same network as SCL:
   "PCS_1".xMod3FltSt := ("PCS_1".wMod3Flt1 <> 0) OR ("PCS_1".wMod3Flt2 <> 0) OR ("PCS_1".wMod3Flt3 <> 0) OR ("PCS_1".wMod3Flt4 <> 0);
END_REGION

REGION Network 26: Inverter Module 4 Fault
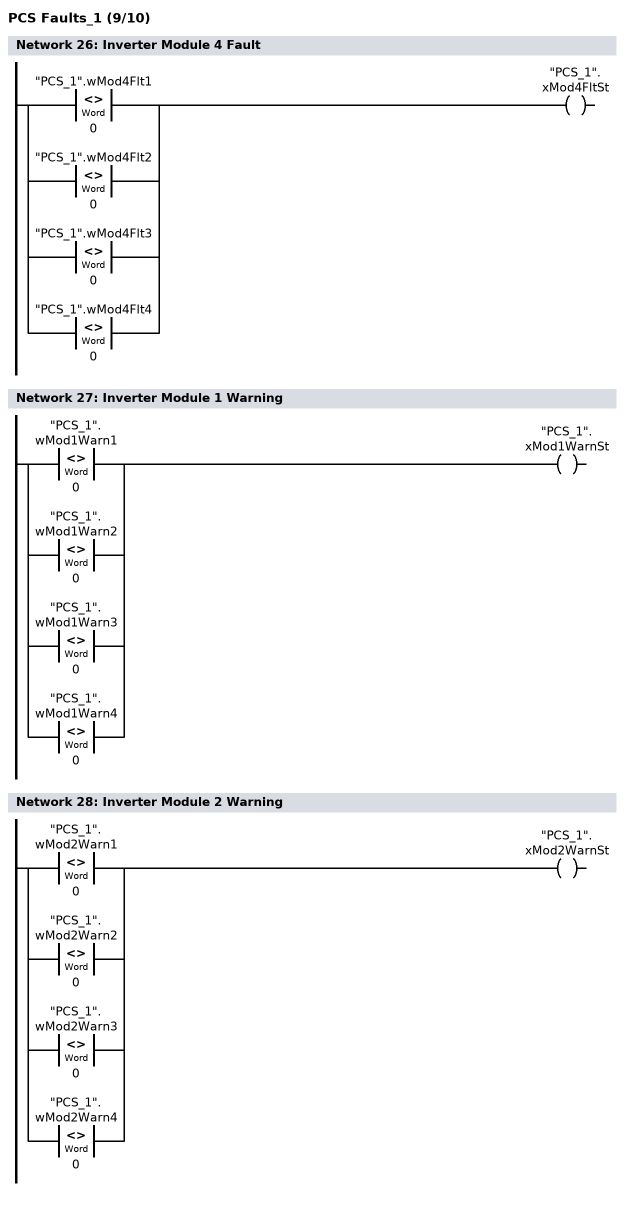
   RUNG wire#powerrail
      { S7_Templates := "SrcType := Word" } NE_Contact(in1 := "PCS_1".wMod4Flt1, in2 := 0)
      wire#w1
      Coil( "PCS_1".xMod4FltSt )
   END_RUNG
   RUNG wire#powerrail
      { S7_Templates := "SrcType := Word" } NE_Contact(in1 := "PCS_1".wMod4Flt2, in2 := 0)
   END_RUNG wire#w1
   RUNG wire#powerrail
      { S7_Templates := "SrcType := Word" } NE_Contact(in1 := "PCS_1".wMod4Flt3, in2 := 0)
   END_RUNG wire#w1
   RUNG wire#powerrail
      { S7_Templates := "SrcType := Word" } NE_Contact(in1 := "PCS_1".wMod4Flt4, in2 := 0)
   END_RUNG wire#w1
   // the same network as SCL:
   "PCS_1".xMod4FltSt := ("PCS_1".wMod4Flt1 <> 0) OR ("PCS_1".wMod4Flt2 <> 0) OR ("PCS_1".wMod4Flt3 <> 0) OR ("PCS_1".wMod4Flt4 <> 0);
END_REGION

REGION Network 27: Inverter Module 1 Warning
   RUNG wire#powerrail
      { S7_Templates := "SrcType := Word" } NE_Contact(in1 := "PCS_1".wMod1Warn1, in2 := 0)
      wire#w1
      Coil( "PCS_1".xMod1WarnSt )
   END_RUNG
   RUNG wire#powerrail
      { S7_Templates := "SrcType := Word" } NE_Contact(in1 := "PCS_1".wMod1Warn2, in2 := 0)
   END_RUNG wire#w1
   RUNG wire#powerrail
      { S7_Templates := "SrcType := Word" } NE_Contact(in1 := "PCS_1".wMod1Warn3, in2 := 0)
   END_RUNG wire#w1
   RUNG wire#powerrail
      { S7_Templates := "SrcType := Word" } NE_Contact(in1 := "PCS_1".wMod1Warn4, in2 := 0)
   END_RUNG wire#w1
   // the same network as SCL:
   "PCS_1".xMod1WarnSt := ("PCS_1".wMod1Warn1 <> 0) OR ("PCS_1".wMod1Warn2 <> 0) OR ("PCS_1".wMod1Warn3 <> 0) OR ("PCS_1".wMod1Warn4 <> 0);
END_REGION

REGION Network 28: Inverter Module 2 Warning
   RUNG wire#powerrail
      { S7_Templates := "SrcType := Word" } NE_Contact(in1 := "PCS_1".wMod2Warn1, in2 := 0)
      wire#w1
      Coil( "PCS_1".xMod2WarnSt )
   END_RUNG
   RUNG wire#powerrail
      { S7_Templates := "SrcType := Word" } NE_Contact(in1 := "PCS_1".wMod2Warn2, in2 := 0)
   END_RUNG wire#w1
   RUNG wire#powerrail
      { S7_Templates := "SrcType := Word" } NE_Contact(in1 := "PCS_1".wMod2Warn3, in2 := 0)
   END_RUNG wire#w1
   RUNG wire#powerrail
      { S7_Templates := "SrcType := Word" } NE_Contact(in1 := "PCS_1".wMod2Warn4, in2 := 0)
   END_RUNG wire#w1
   // the same network as SCL:
   "PCS_1".xMod2WarnSt := ("PCS_1".wMod2Warn1 <> 0) OR ("PCS_1".wMod2Warn2 <> 0) OR ("PCS_1".wMod2Warn3 <> 0) OR ("PCS_1".wMod2Warn4 <> 0);
END_REGION

REGION Network 29: Inverter Module 3 Warning
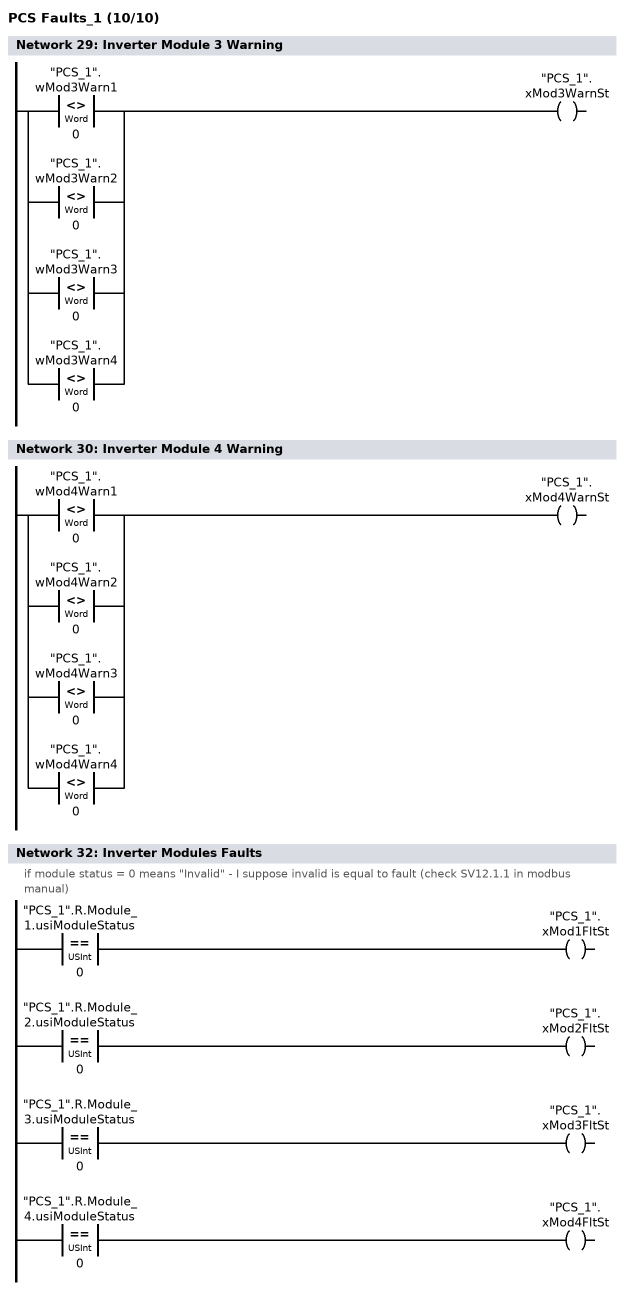
   RUNG wire#powerrail
      { S7_Templates := "SrcType := Word" } NE_Contact(in1 := "PCS_1".wMod3Warn1, in2 := 0)
      wire#w1
      Coil( "PCS_1".xMod3WarnSt )
   END_RUNG
   RUNG wire#powerrail
      { S7_Templates := "SrcType := Word" } NE_Contact(in1 := "PCS_1".wMod3Warn2, in2 := 0)
   END_RUNG wire#w1
   RUNG wire#powerrail
      { S7_Templates := "SrcType := Word" } NE_Contact(in1 := "PCS_1".wMod3Warn3, in2 := 0)
   END_RUNG wire#w1
   RUNG wire#powerrail
      { S7_Templates := "SrcType := Word" } NE_Contact(in1 := "PCS_1".wMod3Warn4, in2 := 0)
   END_RUNG wire#w1
   // the same network as SCL:
   "PCS_1".xMod3WarnSt := ("PCS_1".wMod3Warn1 <> 0) OR ("PCS_1".wMod3Warn2 <> 0) OR ("PCS_1".wMod3Warn3 <> 0) OR ("PCS_1".wMod3Warn4 <> 0);
END_REGION

REGION Network 30: Inverter Module 4 Warning
   RUNG wire#powerrail
      { S7_Templates := "SrcType := Word" } NE_Contact(in1 := "PCS_1".wMod4Warn1, in2 := 0)
      wire#w1
      Coil( "PCS_1".xMod4WarnSt )
   END_RUNG
   RUNG wire#powerrail
      { S7_Templates := "SrcType := Word" } NE_Contact(in1 := "PCS_1".wMod4Warn2, in2 := 0)
   END_RUNG wire#w1
   RUNG wire#powerrail
      { S7_Templates := "SrcType := Word" } NE_Contact(in1 := "PCS_1".wMod4Warn3, in2 := 0)
   END_RUNG wire#w1
   RUNG wire#powerrail
      { S7_Templates := "SrcType := Word" } NE_Contact(in1 := "PCS_1".wMod4Warn4, in2 := 0)
   END_RUNG wire#w1
   // the same network as SCL:
   "PCS_1".xMod4WarnSt := ("PCS_1".wMod4Warn1 <> 0) OR ("PCS_1".wMod4Warn2 <> 0) OR ("PCS_1".wMod4Warn3 <> 0) OR ("PCS_1".wMod4Warn4 <> 0);
END_REGION

REGION Network 31: -> Fine OLD
END_REGION

REGION Network 32: Inverter Modules Faults
   // if module status = 0 means "Invalid" - I suppose invalid is equal to fault (check SV12.1.1 in modbus manual)
   RUNG wire#powerrail
      { S7_Templates := "SrcType := USInt" } EQ_Contact(in1 := "PCS_1".R.Module_1.usiModuleStatus, in2 := 0)
      Coil( "PCS_1".xMod1FltSt )
   END_RUNG
   RUNG wire#powerrail
      { S7_Templates := "SrcType := USInt" } EQ_Contact(in1 := "PCS_1".R.Module_2.usiModuleStatus, in2 := 0)
      Coil( "PCS_1".xMod2FltSt )
   END_RUNG
   RUNG wire#powerrail
      { S7_Templates := "SrcType := USInt" } EQ_Contact(in1 := "PCS_1".R.Module_3.usiModuleStatus, in2 := 0)
      Coil( "PCS_1".xMod3FltSt )
   END_RUNG
   RUNG wire#powerrail
      { S7_Templates := "SrcType := USInt" } EQ_Contact(in1 := "PCS_1".R.Module_4.usiModuleStatus, in2 := 0)
      Coil( "PCS_1".xMod4FltSt )
   END_RUNG
   // the same network as SCL:
   "PCS_1".xMod1FltSt := "PCS_1".R.Module_1.usiModuleStatus = 0;
   "PCS_1".xMod2FltSt := "PCS_1".R.Module_2.usiModuleStatus = 0;
   "PCS_1".xMod3FltSt := "PCS_1".R.Module_3.usiModuleStatus = 0;
   "PCS_1".xMod4FltSt := "PCS_1".R.Module_4.usiModuleStatus = 0;
END_REGION
END_FUNCTION
